TYPE ST_SafetyFB :
STRUCT
    sName : STRING;
    Diag AT %I* : UINT;
    State AT %I* : USINT;
    eFbType : E_SafetyFbType;
    fbState : E_SafetyFbState;
    DiagString : STRING;
END_STRUCT
END_TYPE

(* stored: Version 1.1.0.1, ProductVersion 3.1.4024.11
   DUT ST_SafetyFB: Id {99c96ab4-3a2f-494f-8007-18f6e4529433} *)
